// TIA Portal V20 export
TYPE "LER_typeCommunicationBSENDCommands"
// stored: Access Published
   STRUCT
      req : Bool;
      reset : Bool;
   END_STRUCT;
END_TYPE
